// Mitsubishi GX Works2 project: 0709   PLC: Q02/Q02H

PROGRAM MAIN
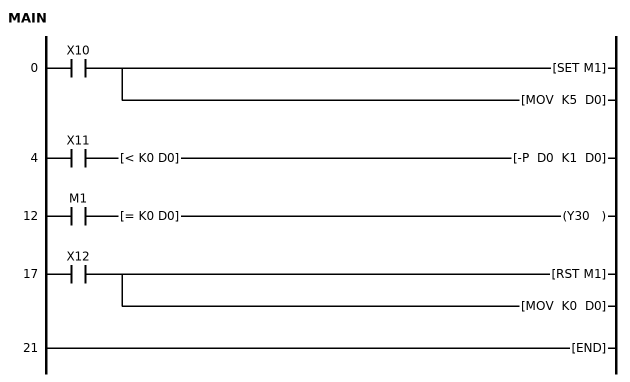
0     LD      X10
      SET     M1
      MOV     K5 D0
4     LD      X11
      AND<    K0 D0
      -P      D0 K1 D0
12    LD      M1
      AND=    K0 D0
      OUT     Y30
17    LD      X12
      RST     M1
      MOV     K0 D0
21    END
END_PROGRAM

PROGRAM MAIN1
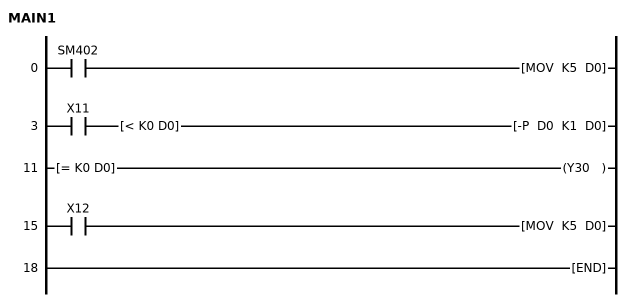
0     LD      SM402
      MOV     K5 D0
3     LD      X11
      AND<    K0 D0
      -P      D0 K1 D0
11    LD=     K0 D0
      OUT     Y30
15    LD      X12
      MOV     K5 D0
18    END
END_PROGRAM

PROGRAM MAIN2
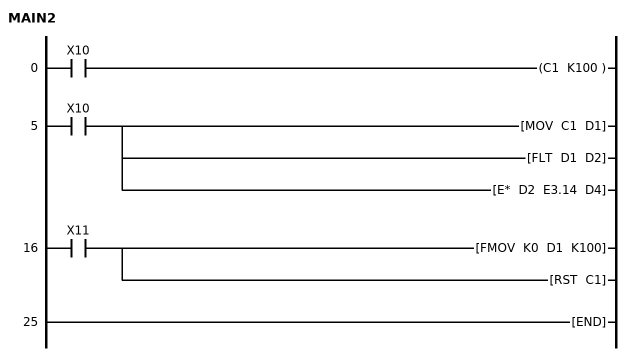
0     LD      X10
      OUT     C1 K100
5     LD      X10
      MOV     C1 D1
      FLT     D1 D2
      E*      D2 E3.14 D4
16    LD      X11
      FMOV    K0 D1 K100
      RST     C1
25    END
END_PROGRAM

PROGRAM MAIN3
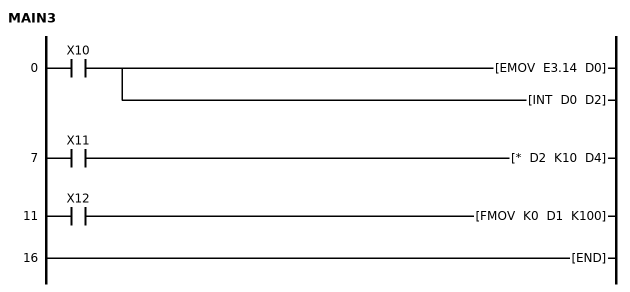
0     LD      X10
      EMOV    E3.14 D0
      INT     D0 D2
7     LD      X11
      *       D2 K10 D4
11    LD      X12
      FMOV    K0 D1 K100
16    END
END_PROGRAM

PROGRAM MAIN4
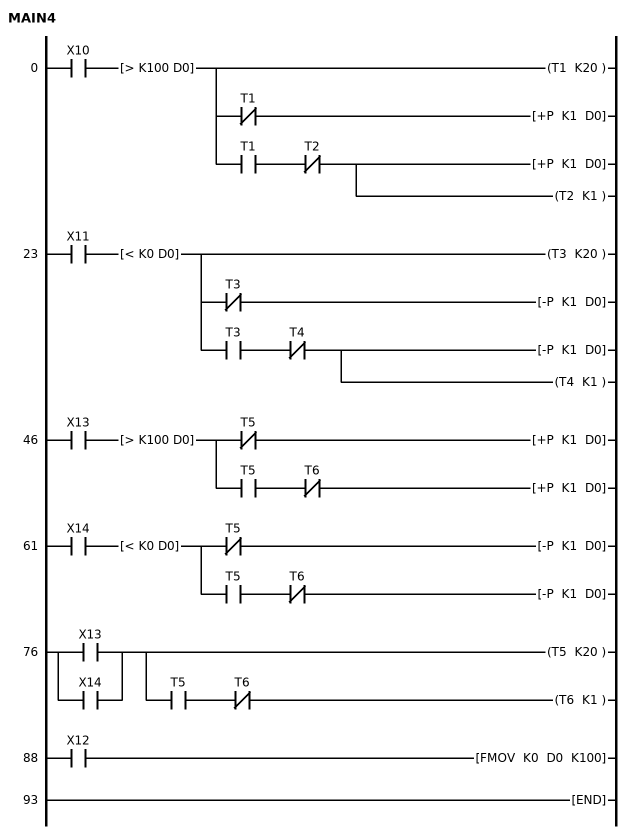
0     LD      X10
      AND>    K100 D0
      OUT     T1 K20
      MPS
      ANI     T1
      +P      K1 D0
      MPP
      AND     T1
      ANI     T2
      +P      K1 D0
      OUT     T2 K1
23    LD      X11
      AND<    K0 D0
      OUT     T3 K20
      MPS
      ANI     T3
      -P      K1 D0
      MPP
      AND     T3
      ANI     T4
      -P      K1 D0
      OUT     T4 K1
46    LD      X13
      AND>    K100 D0
      MPS
      ANI     T5
      +P      K1 D0
      MPP
      AND     T5
      ANI     T6
      +P      K1 D0
61    LD      X14
      AND<    K0 D0
      MPS
      ANI     T5
      -P      K1 D0
      MPP
      AND     T5
      ANI     T6
      -P      K1 D0
76    LD      X13
      OR      X14
      OUT     T5 K20
      AND     T5
      ANI     T6
      OUT     T6 K1
88    LD      X12
      FMOV    K0 D0 K100
93    END
END_PROGRAM

PROGRAM MAIN5
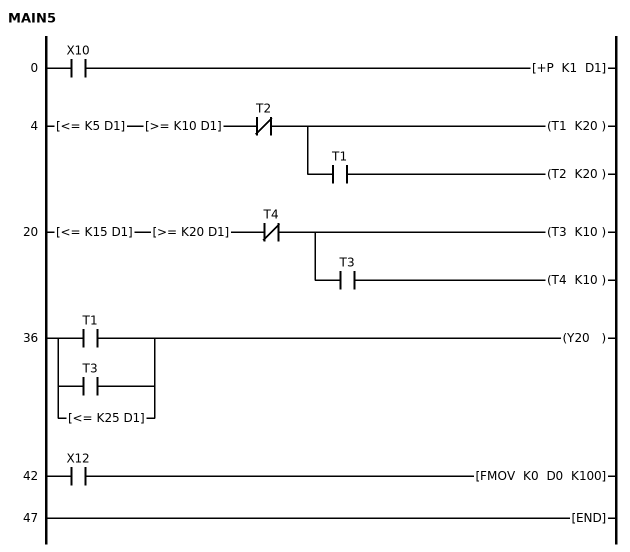
0     LD      X10
      +P      K1 D1
4     LD<=    K5 D1
      AND>=   K10 D1
      ANI     T2
      OUT     T1 K20
      AND     T1
      OUT     T2 K20
20    LD<=    K15 D1
      AND>=   K20 D1
      ANI     T4
      OUT     T3 K10
      AND     T3
      OUT     T4 K10
36    LD      T1
      OR      T3
      OR<=    K25 D1
      OUT     Y20
42    LD      X12
      FMOV    K0 D0 K100
47    END
END_PROGRAM

PROGRAM MAIN6
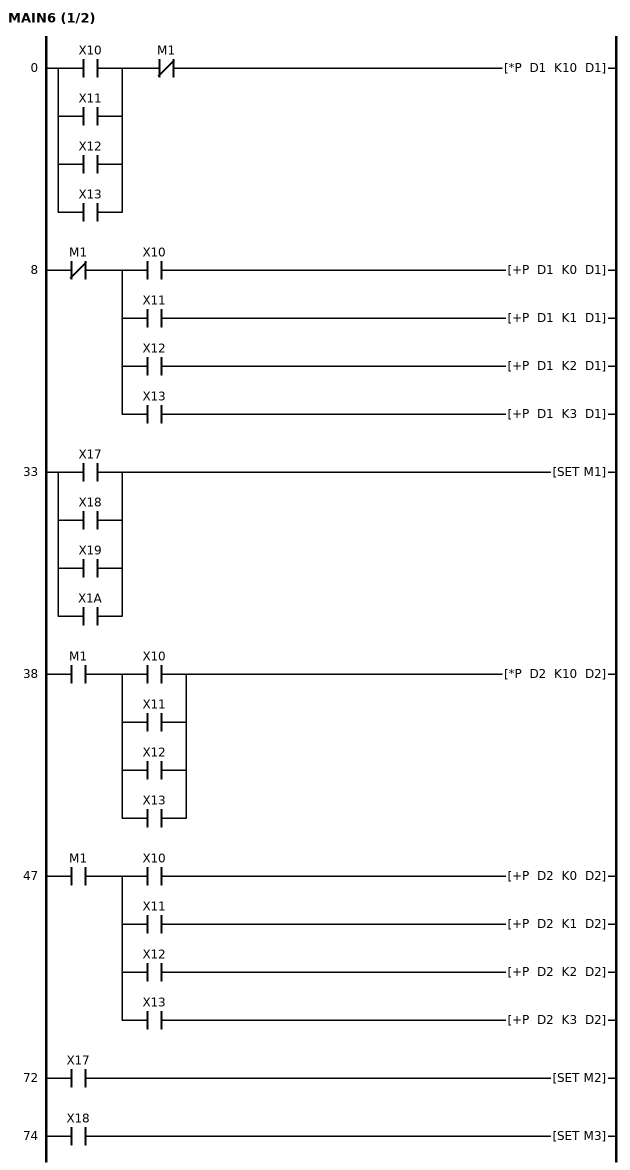
0     LD      X10
      OR      X11
      OR      X12
      OR      X13
      ANI     M1
      *P      D1 K10 D1
8     LDI     M1
      MPS
      AND     X10
      +P      D1 K0 D1
      MRD
      AND     X11
      +P      D1 K1 D1
      MRD
      AND     X12
      +P      D1 K2 D1
      MPP
      AND     X13
      +P      D1 K3 D1
33    LD      X17
      OR      X18
      OR      X19
      OR      X1A
      SET     M1
38    LD      M1
      LD      X10
      OR      X11
      OR      X12
      OR      X13
      ANB
      *P      D2 K10 D2
47    LD      M1
      MPS
      AND     X10
      +P      D2 K0 D2
      MRD
      AND     X11
      +P      D2 K1 D2
      MRD
      AND     X12
      +P      D2 K2 D2
      MPP
      AND     X13
      +P      D2 K3 D2
72    LD      X17
      SET     M2
74    LD      X18
      SET     M3
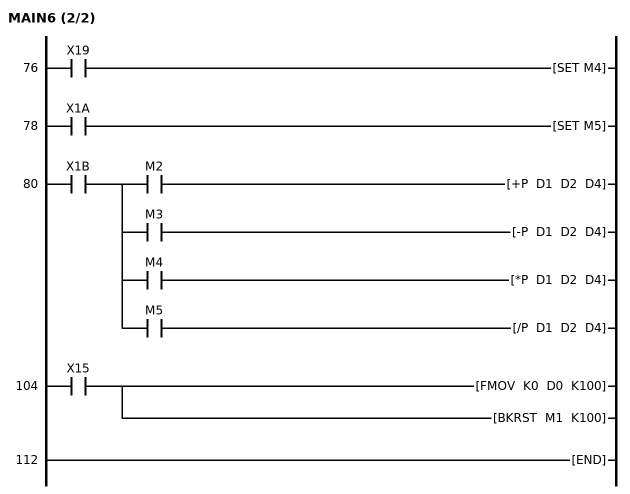
76    LD      X19
      SET     M4
78    LD      X1A
      SET     M5
80    LD      X1B
      MPS
      AND     M2
      +P      D1 D2 D4
      MRD
      AND     M3
      -P      D1 D2 D4
      MRD
      AND     M4
      *P      D1 D2 D4
      MPP
      AND     M5
      /P      D1 D2 D4
104   LD      X15
      FMOV    K0 D0 K100
      BKRST   M1 K100
112   END
END_PROGRAM

PROGRAM MAIN7
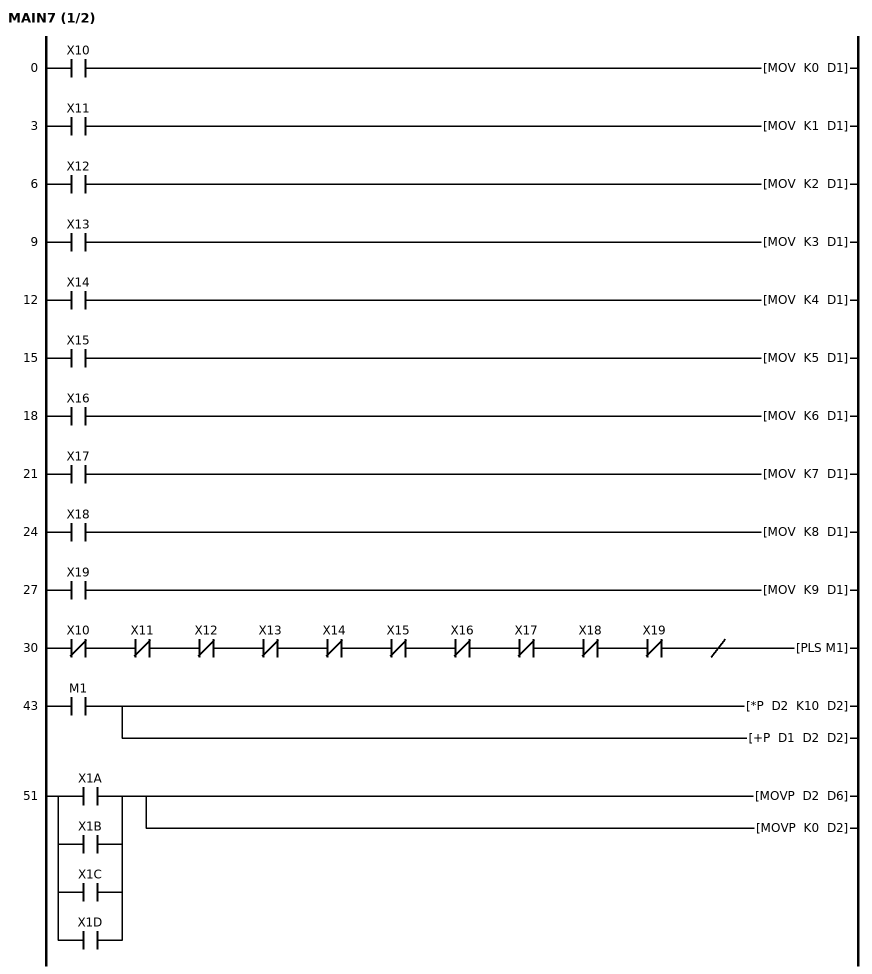
0     LD      X10
      MOV     K0 D1
3     LD      X11
      MOV     K1 D1
6     LD      X12
      MOV     K2 D1
9     LD      X13
      MOV     K3 D1
12    LD      X14
      MOV     K4 D1
15    LD      X15
      MOV     K5 D1
18    LD      X16
      MOV     K6 D1
21    LD      X17
      MOV     K7 D1
24    LD      X18
      MOV     K8 D1
27    LD      X19
      MOV     K9 D1
30    LDI     X10
      ANI     X11
      ANI     X12
      ANI     X13
      ANI     X14
      ANI     X15
      ANI     X16
      ANI     X17
      ANI     X18
      ANI     X19
      INV
      PLS     M1
43    LD      M1
      *P      D2 K10 D2
      +P      D1 D2 D2
51    LD      X1A
      OR      X1B
      OR      X1C
      OR      X1D
      MOVP    D2 D6
      MOVP    K0 D2
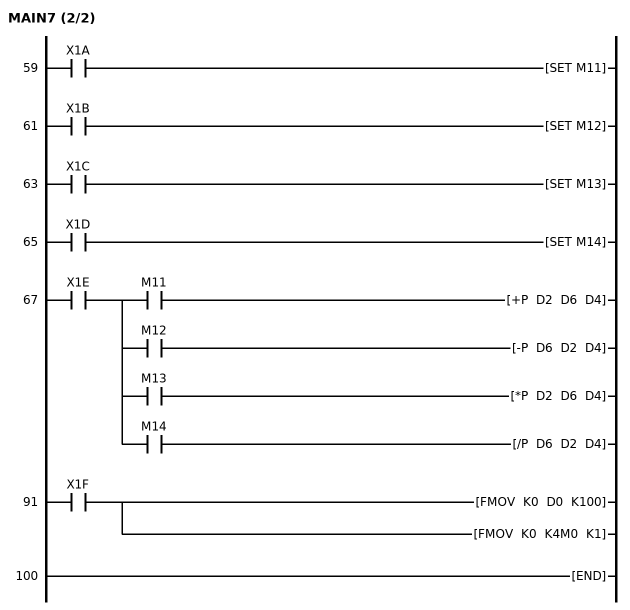
59    LD      X1A
      SET     M11
61    LD      X1B
      SET     M12
63    LD      X1C
      SET     M13
65    LD      X1D
      SET     M14
67    LD      X1E
      MPS
      AND     M11
      +P      D2 D6 D4
      MRD
      AND     M12
      -P      D6 D2 D4
      MRD
      AND     M13
      *P      D2 D6 D4
      MPP
      AND     M14
      /P      D6 D2 D4
91    LD      X1F
      FMOV    K0 D0 K100
      FMOV    K0 K4M0 K1
100   END
END_PROGRAM
